FUNCTION_BLOCK ABBScannerStation
VAR_INPUT
	mxEnable: BOOL;
END_VAR
VAR_OUTPUT
	mxDone:BOOL;
	mxExecuting: BOOL;
	mxError: BOOL;
END_VAR
VAR
	ABB: INT;
	mxWaitingforsensorinput: BOOL;
END_VAR

CASE ABB OF
	0:
		IF mxEnable THEN
			ABB:=10;
		END_IF
	10:
		IF (CommData.mwXaxis = CommData.ABBPostions.Scannerhome.X AND CommData.mwYaxis = CommData.ABBPostions.Scannerhome.Y) OR CommData.msRobotLastPos = 'Scanner'  THEN
			ABB:=20;
		ELSIF CommData.mxRobotOnline THEN
			ABB:=30;
		ELSE
			ABB:=1000;
		END_IF
	20:
		IF CommData.mxRobotOnline THEN
			ABB:=30;
		ELSE
			mxExecuting:=TRUE;
			commdata.mxWaitingforSensorinput:=TRUE;
			IF CommData.mxScannernoobject THEN
				ABB:=30;
			END_IF
		END_IF	
	30:
		commdata.mxWaitingforSensorinput:=FALSE;
		mxExecuting:=FALSE;
		mxDone:=TRUE;
		IF NOT mxEnable THEN
			mxDone:=FALSE;
			ABB:=0;
		END_IF
	1000:
		mxExecuting:=FALSE;
		mxError:=TRUE;
		IF NOT mxEnable THEN
			mxError:=FALSE;
			mxDone:=FALSE;
			ABB:=0;
		END_IF
		
END_CASE



IF gvl.ixEmergencyStop THEN
	ABB:=1000;
END_IF

END_FUNCTION_BLOCK

(* stored: Version 1.1.0.1, ProductVersion 3.1.4024.12
   POU ABBScannerStation: Id {41bb971a-3d77-47a0-9f8d-97aedaa7a92a}, SpecialFunc None *)
